// TIA Portal V16 export
// export: Created 2021-07-12T14:47:19.1457318Z, ExportSetting WithDefaults, DisplayName Totally Integrated Automation Portal, DisplayVersion V16, DisplayName TIA Portal Version Control Interface, DisplayVersion V16, DisplayName TIA Portal Openness, DisplayVersion V16, DisplayName STEP 7 Professional, DisplayVersion V16, DisplayName STEP 7 Safety, DisplayVersion V16, DisplayName WinCC Professional, DisplayVersion V16
TYPE "LSimaHydTO_typePositionLimits"
TITLE = LSimaHydTO_typePositionLimits
// Software position limit switch
// stored: IsFailsafeCompliant false
   STRUCT
      Active { S7_SetPoint := 'True'} : Bool := TRUE;   // FALSE: Monitoring disabled / TRUE: Monitoring enabled
      MinPosition { S7_SetPoint := 'True'} : LReal := -1000000000000.0;   // Position of negative SW limit switch
      MaxPosition { S7_SetPoint := 'True'} : LReal := 1000000000000.0;   // Position of positive SW limit switch
   END_STRUCT;
END_TYPE
